// SIMATIC S7-200 project (STEP 7-Micro/WIN), CPU 221 REL 01.10

ORGANIZATION_BLOCK 启保停法实现:OB1
TITLE=
BEGIN
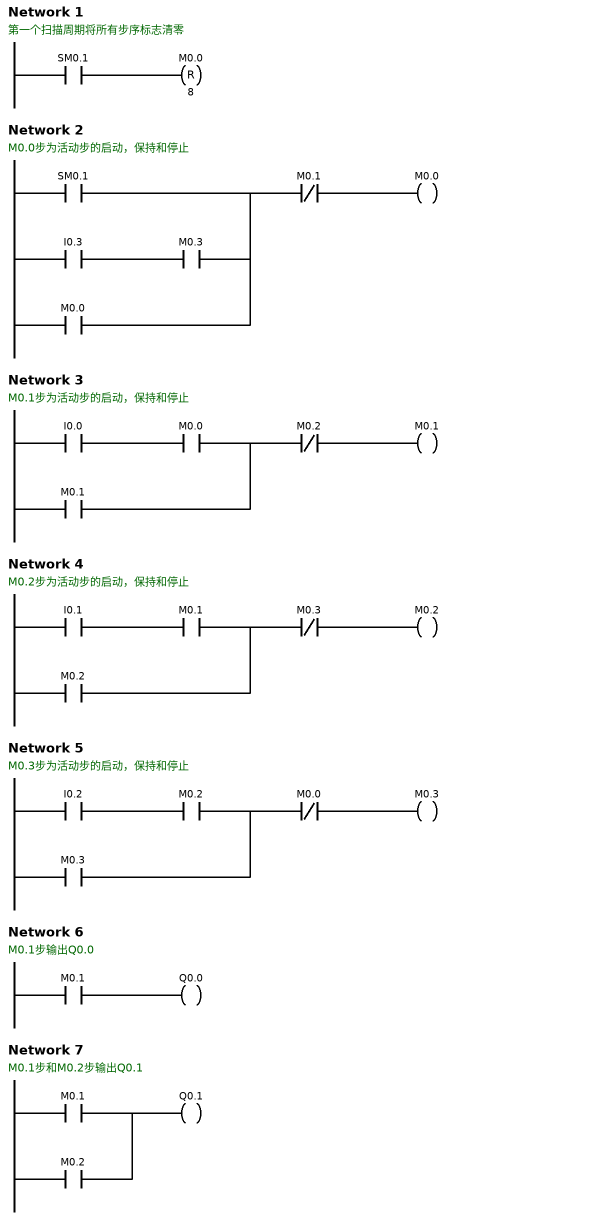
Network 1
// 第一个扫描周期将所有步序标志清零
LD     SM0.1
R      M0.0, 8
Network 2
// M0.0步为活动步的启动，保持和停止
LD     SM0.1
LD     I0.3
A      M0.3
OLD
O      M0.0
AN     M0.1
=      M0.0
Network 3
// M0.1步为活动步的启动，保持和停止
LD     I0.0
A      M0.0
O      M0.1
AN     M0.2
=      M0.1
Network 4
// M0.2步为活动步的启动，保持和停止
// (network saved uncompiled; LAD cells follow)
// row 0: c0 -| |- I0.1  c1 -| |- M0.1 v  c2 -|/|- M0.3  c3 -( ) M0.2
// row 1: c0 -| |- M0.2  c1 -- ^
Network 5
// M0.3步为活动步的启动，保持和停止
// (network saved uncompiled; LAD cells follow)
// row 0: c0 -| |- I0.2  c1 -| |- M0.2 v  c2 -|/|- M0.0  c3 -( ) M0.3
// row 1: c0 -| |- M0.3  c1 -- ^
Network 6
// M0.1步输出Q0.0
// (network saved uncompiled; LAD cells follow)
// row 0: c0 -| |- M0.1  c1 -( ) Q0.0
Network 7
// M0.1步和M0.2步输出Q0.1
// (network saved uncompiled; LAD cells follow)
// row 0: c0 -| |- M0.1 v  c1 -( ) Q0.1
// row 1: c0 -| |- M0.2 ^
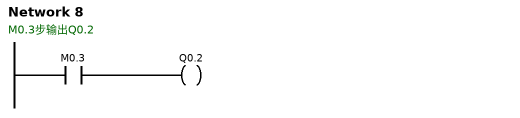
Network 8
// M0.3步输出Q0.2
// (network saved uncompiled; LAD cells follow)
// row 0: c0 -| |- M0.3  c1 -( ) Q0.2
END_ORGANIZATION_BLOCK

SUBROUTINE_BLOCK 置位复位法实现:SBR0
TITLE=
BEGIN
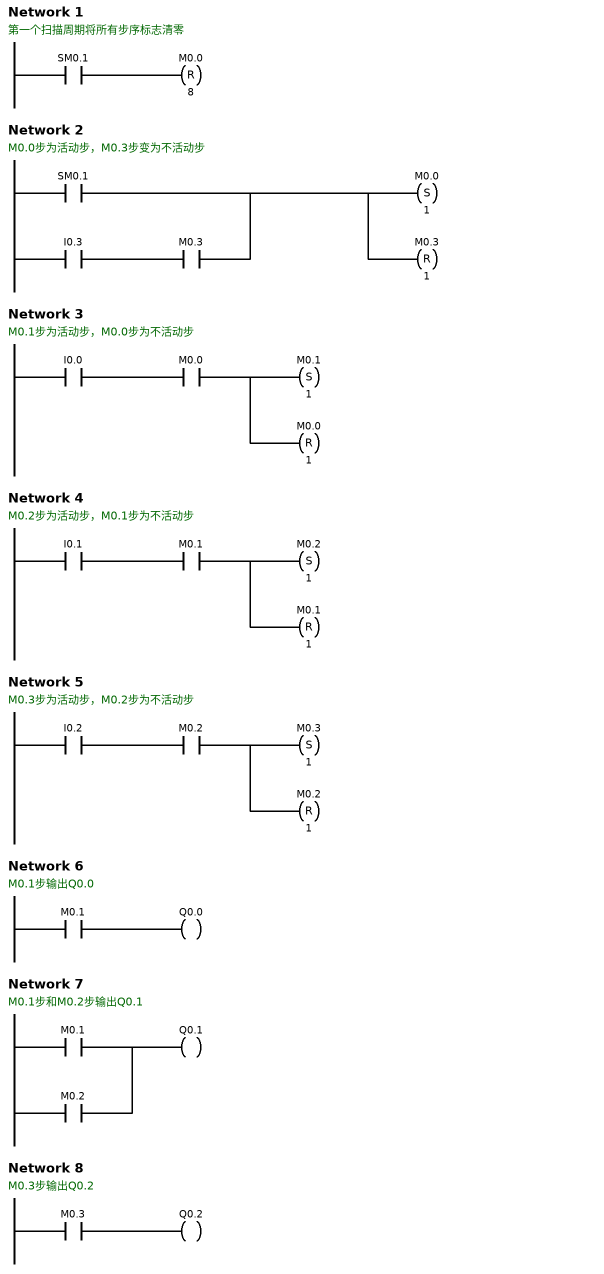
Network 1
// 第一个扫描周期将所有步序标志清零
LD     SM0.1
R      M0.0, 8
Network 2
// M0.0步为活动步，M0.3步变为不活动步
// (network saved uncompiled; LAD cells follow)
// row 0: c0 -| |- SM0.1  c1 -- v  c2 -- v  c3 -(S) M0.0, 1
// row 1: c0 -| |- I0.3  c1 -| |- M0.3 ^  c2 ^  c3 -(R) M0.3, 1
Network 3
// M0.1步为活动步，M0.0步为不活动步
// (network saved uncompiled; LAD cells follow)
// row 0: c0 -| |- I0.0  c1 -| |- M0.0 v  c2 -(S) M0.1, 1
// row 1: c1 ^  c2 -(R) M0.0, 1
Network 4
// M0.2步为活动步，M0.1步为不活动步
// (network saved uncompiled; LAD cells follow)
// row 0: c0 -| |- I0.1  c1 -| |- M0.1 v  c2 -(S) M0.2, 1
// row 1: c1 ^  c2 -(R) M0.1, 1
Network 5
// M0.3步为活动步，M0.2步为不活动步
// (network saved uncompiled; LAD cells follow)
// row 0: c0 -| |- I0.2  c1 -| |- M0.2 v  c2 -(S) M0.3, 1
// row 1: c1 ^  c2 -(R) M0.2, 1
Network 6
// M0.1步输出Q0.0
LD     M0.1
=      Q0.0
Network 7
// M0.1步和M0.2步输出Q0.1
LD     M0.1
O      M0.2
=      Q0.1
Network 8
// M0.3步输出Q0.2
LD     M0.3
=      Q0.2
END_SUBROUTINE_BLOCK

INTERRUPT_BLOCK SCR指令实现:INT0
TITLE=
BEGIN
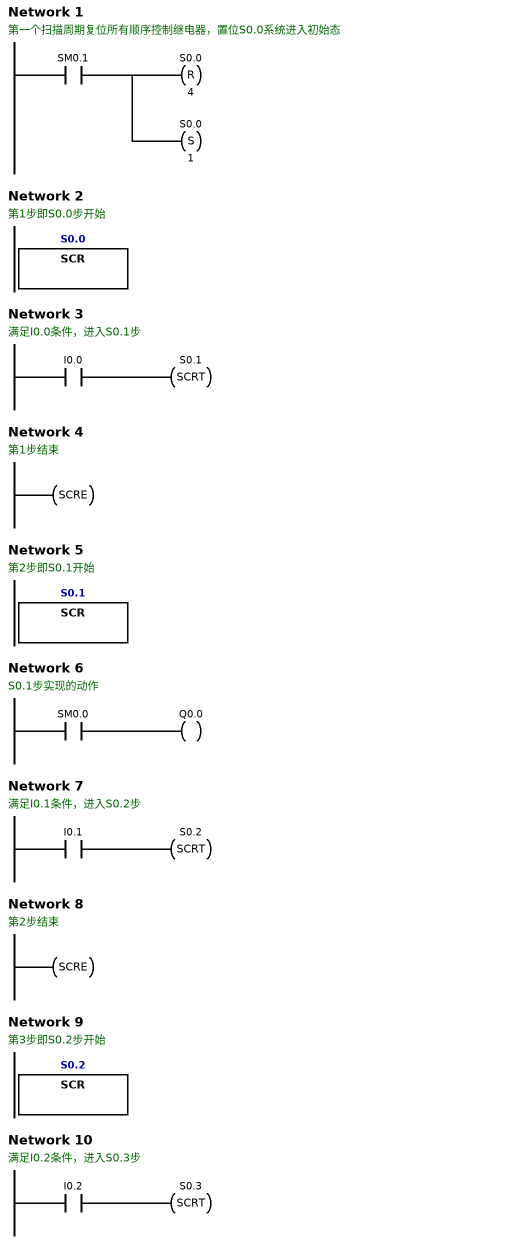
Network 1
// 第一个扫描周期复位所有顺序控制继电器，置位S0.0系统进入初始态
// (network saved uncompiled; LAD cells follow)
// row 0: c0 -| |- SM0.1 v  c1 -(R) S0.0, 4
// row 1: c0 ^  c1 -(S) S0.0, 1
Network 2
// 第1步即S0.0步开始
// (network saved uncompiled; LAD cells follow)
// row 0: c0 [SCR S0.0 ]
Network 3
// 满足I0.0条件，进入S0.1步
// (network saved uncompiled; LAD cells follow)
// row 0: c0 -| |- I0.0  c1 -(SCRT) S0.1
Network 4
// 第1步结束
// (network saved uncompiled; LAD cells follow)
// row 0: c0 -(SCRE)
Network 5
// 第2步即S0.1开始
// (network saved uncompiled; LAD cells follow)
// row 0: c0 [SCR S0.1 ]
Network 6
// S0.1步实现的动作
// (network saved uncompiled; LAD cells follow)
// row 0: c0 -| |- SM0.0  c1 -( ) Q0.0
Network 7
// 满足I0.1条件，进入S0.2步
// (network saved uncompiled; LAD cells follow)
// row 0: c0 -| |- I0.1  c1 -(SCRT) S0.2
Network 8
// 第2步结束
// (network saved uncompiled; LAD cells follow)
// row 0: c0 -(SCRE)
Network 9
// 第3步即S0.2步开始
// (network saved uncompiled; LAD cells follow)
// row 0: c0 [SCR S0.2 ]
Network 10
// 满足I0.2条件，进入S0.3步
// (network saved uncompiled; LAD cells follow)
// row 0: c0 -| |- I0.2  c1 -(SCRT) S0.3
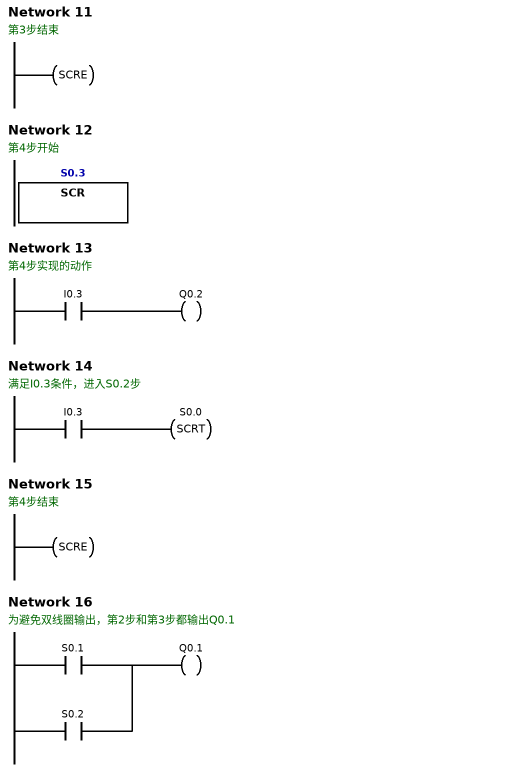
Network 11
// 第3步结束
// (network saved uncompiled; LAD cells follow)
// row 0: c0 -(SCRE)
Network 12
// 第4步开始
// (network saved uncompiled; LAD cells follow)
// row 0: c0 [SCR S0.3 ]
Network 13
// 第4步实现的动作
// (network saved uncompiled; LAD cells follow)
// row 0: c0 -| |- I0.3  c1 -( ) Q0.2
Network 14
// 满足I0.3条件，进入S0.2步
// (network saved uncompiled; LAD cells follow)
// row 0: c0 -| |- I0.3  c1 -(SCRT) S0.0
Network 15
// 第4步结束
// (network saved uncompiled; LAD cells follow)
// row 0: c0 -(SCRE)
Network 16
// 为避免双线圈输出，第2步和第3步都输出Q0.1
// (network saved uncompiled; LAD cells follow)
// row 0: c0 -| |- S0.1 v  c1 -( ) Q0.1
// row 1: c0 -| |- S0.2 ^
END_INTERRUPT_BLOCK
